FUNCTION_BLOCK Heating_OnRequest IMPLEMENTS I_Callable
VAR
	_ctx			: REFERENCE TO Heating_Ctx;
END_VAR

METHOD Call
VAR_INPUT
	iArg				: Core.I_Arg;
END_VAR
VAR
	_iRoom				: I_Room;
END_VAR
IF IsOk(IArgToIRoom(iArg, iDest => _iRoom)) THEN
	_ctx.priv.iQueue.Push(_iRoom);
END_IF
END_METHOD

//FB_Init is always available implicitly and it is used primarily for initialization.
//The return value is not evaluated. For a specific influence, you can also declare the
//methods explicitly and provide additional code there with the standard initialization
//code. You can evaluate the return value.
METHOD FB_Init: BOOL
VAR_INPUT
    bInitRetains: BOOL; // TRUE: the retain variables are initialized (reset warm / reset cold)
    bInCopyCode: BOOL;  // TRUE: the instance will be copied to the copy code afterward (online change)

	ctx			: REFERENCE TO Heating_Ctx;   
END_VAR
_ctx REF= ctx;
END_METHOD

END_FUNCTION_BLOCK

(* stored: Version 1.1.0.1
   POU Heating_OnRequest: Id {f1fcf00f-bece-4c8c-95ed-661830145846}, SpecialFunc None
   Method Call: Id {d2f41e16-5d62-432c-8cbc-b541da0bb20b}
   Method FB_init: Id {58f7fbb6-9133-4052-9821-9af265dc0ec8} *)
